FUNCTION_BLOCK CONTROL_ITER
  (* Standard: 61499-2 *)
  (* Version 1.0, 31/05/2012, GASR *)
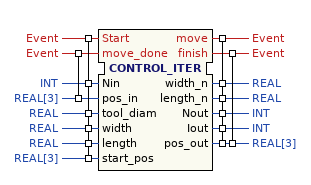
  EVENT_INPUT
    Start WITH width, length, start_pos, Nin, tool_diam; (* first time execution *)
    move_done WITH pos_in;
  END_EVENT
  EVENT_OUTPUT
    move WITH width_n, length_n, pos_out, Iout, Nout, start_pos, tool_diam;
    finish WITH pos_out;
  END_EVENT
  VAR_INPUT
    Nin : INT;
    pos_in : ARRAY [0..2] OF REAL;
    tool_diam : REAL;
    width : REAL;
    length : REAL;
    start_pos : ARRAY [0..2] OF REAL;
  END_VAR
  VAR_OUTPUT
    width_n : REAL;
    length_n : REAL;
    Nout : INT;
    Iout : INT;
    pos_out : ARRAY [0..2] OF REAL;
  END_VAR
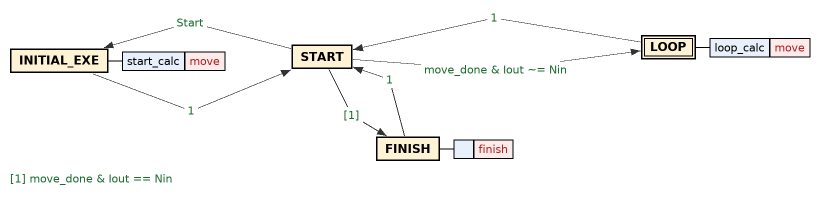
  EC_STATES
    LOOP : loop_calc -> move;
    START;
    FINISH : -> finish;
    INITIAL_EXE : start_calc -> move;
  END_STATES
  EC_TRANSITIONS
    START TO INITIAL_EXE := Start;
    START TO LOOP := move_done & Iout ~= Nin;
    START TO FINISH := move_done & Iout == Nin;
    LOOP TO START := 1;
    INITIAL_EXE TO START := 1;
    FINISH TO START := 1;
  END_TRANSITIONS
  ALGORITHM start_calc IN Lua:
        width_n = tonumber(width-tool_diam)    length_n = tonumber(length - tool_diam)    pos_out = {start_pos[1],start_pos[2], start_pos[3]}     Iout = 0    Nout = Nin
  END_ALGORITHM
  ALGORITHM loop_calc IN Lua:
    Iout = Iout + 1    width_n = ((Nin-Iout)/Nin)*(width -tool_diam)    length_n = ((Nin-Iout)/Nin)*(length-tool_diam)    Nout = Nin    pos_out = {pos_in[1], pos_in[2], pos_in[3]}
  END_ALGORITHM
END_FUNCTION_BLOCK
